//==================================================================================================
//							Beckhoff Automation Poland
//									19.09.2017
// Procedura restartu - najpierw grupa, pozniej karta, na koncu bloki
// Uwaga - w przypadku bledu grupy, bledy karty nie sa widoczne jeszce przez chwile po resecie grupy.
// Dlatego dodane jest opoznienie
//	v1.0 	|| TC v 3.1.4022.2 || - pierwsza wersja
//==================================================================================================
PROGRAM P_SAFETY
VAR
	iStep						: INT;
	tonDelay					: TON;
	bDelayReq					: BOOL;
	tonDelay2: TON;
	tonDelay3: TON;
END_VAR

tonDelay.IN 								:= iStep = 10 OR iStep = 40;
tonDelay.PT									:= T#300MS;
tonDelay();

tonDelay2.IN								:= iStep = 20;
tonDelay2.PT								:= T#100MS;
tonDelay2();

tonDelay3.IN								:= iStep = 30;
tonDelay3.PT								:= T#3000MS;
tonDelay3();
//flagi błędu komunikacji
QbCommunicationErrorUP50B					:= (IbComErr_Gr2 OR IbFBErr_Gr2 OR IbOtherErr_Gr2 OR NOT IbOutErr_Gr2) AND NOT IbUP50BDeactivated;
QbCommunicationErrorUF50					:= (IbComErr_Gr3 OR IbFBErr_Gr3 OR IbOtherErr_Gr3 OR NOT IbOutErr_Gr3) AND NOT IbUF50Deactivated;




// Procedura
CASE iStep OF
	
	0: // Oczekiwanie na reset
	IF ((bSafetyResetIn OR IbSafetyResetCapSorterIn OR IbSafetyResetBottleSorterIn OR bPucksInserterSafetyResetIn OR bSafetyResetInRC40) AND
		NOT bEmergencyStop) AND IbSafetyResetDelay //Opóżnieni 30s z UBL tylko przy pierwszym uruchomieniu
	 	THEN
		QbRUN_STOP_GR2				R= IbComErr_Gr2 OR IbFBErr_Gr2 OR IbOtherErr_Gr2 OR NOT IbOutErr_Gr2;
		QbRUN_STOP_GR3				R= IbComErr_Gr3 OR IbFBErr_Gr3 OR IbOtherErr_Gr3 OR NOT IbOutErr_Gr3;
		iStep 						:= iStep + 10;
	END_IF
	
	10:	// Reset bledu grupy - jesli jest
		QbRUN_STOP					:= TRUE;
		//QbRUN_STOP_GR2				R= IbComErr_Gr2 OR IbFBErr_Gr2 OR IbOtherErr_Gr2 OR NOT IbOutErr_Gr2;
		//QbRUN_STOP_GR3				R= IbComErr_Gr3 OR IbFBErr_Gr3 OR IbOtherErr_Gr3 OR NOT IbOutErr_Gr3;
		IF tonDelay.Q THEN
			QbRUN_STOP							:= TRUE;
			QbRUN_STOP_GR2						:= TRUE;
			QbRUN_STOP_GR3						:= TRUE;
			bErrorAck							:= TRUE;
			bErrorAckGr2						:= TRUE;
			bErrorAckGr3						:= TRUE;
			bSafetyReset			:= TRUE;
			bSafetyReset2			:= TRUE;
			iStep 								:= iStep + 10;
		END_IF
	
	20: // Reset bledu karty AX5805 - jesli jest
		IF tonDelay2.Q THEN
			bErrorAck			:= FALSE;
			bErrorAckGr2			:= FALSE;
			bErrorAckGr3			:= FALSE;
			bSafetyReset			:= FALSE;
			bSafetyReset2			:= FALSE;
			bSafetyReset3			:= TRUE;
			iStep 					:= iStep + 10;	
		END_IF
	

	30:
		IF tonDelay3.Q THEN
			bSafetyReset			:= FALSE;
			bSafetyReset2			:= FALSE;
			bSafetyReset3			:= false;
			iStep 					:= iStep + 10;	
		END_IF
	
	40:
		IF tonDelay.Q THEN
			bSafetyReset3			:= FALSE;
			iStep	 				:= 0;
		END_IF
	
END_CASE

END_PROGRAM

(* stored: Version 1.1.0.1, ProductVersion 3.1.4026.13, FileIdentifier bde6bc99b58ffedc5473a8d6ec5a0d8a42c4b453, FileSignature 3976d750caaa2681ceb289e73cabd2cf09e66ae1eaef512a71608756abf6f958fb72acc6125e1b03d3a6b75210d036068f3f2547ed7f9337db2dfa8f9618fcc547356bd8d4d612993f9510bcb0c0e2f0d0d29c587fd28c6e65b976671d54adb908f4e595e12d21793a91a62de9758d252af108505744e8b4c4745a050d1831da0469bbf53f8ad6f74f91e24b4f0398866dddf0edbf562e5a4d14aa7b55714d0301f415a269f9ed21cdb55dfe5472fc9ad75364b511a4592ce7c3b61075892c0e55ca08368ba9e2d138dc292ae845eae8eb42e235c97ff8bfea6a508db0ddb4add0956518732f72a57fbd8c0ff05902e8722f951fa3d25a66a8b8a3dfd13ed0a9
   POU P_SAFETY: Id {72856a85-4209-4393-9c43-65ed18b02966}, SpecialFunc None *)
